(* IEC 61131-3 sources: Lasal/CPU_5344_V01/Class/RestartClass, 1 file *)

(* ---- RestartClass.st ---- *)
(*!
<Class
	Name               = "RestartClass"
	Revision           = "0.0"
	RealtimeTask       = "false"
	CyclicTask         = "false"
	BackgroundTask     = "false"
	Sigmatek           = "false"
	OSInterface        = "false"
	HighPriority       = "false"
	Automatic          = "false"
	UpdateMode         = "Prescan"
	SharedCommandTable = "true"
	Objectsize         = "(284,120)">
	<Channels>
		<Server Name="ClassSvr" Visualized="true" Initialize="false" WriteProtected="false" Retentive="false"/>
		<Client Name="os" Required="false" Internal="false"/>
	</Channels>
</Class>
*)
RestartClass : CLASS
  //Servers:
	ClassSvr 	: SvrChCmd_DINT;
  //Clients:
	os 	: CltChCmd__OSKernel;
  //Variables:
  //Functions:

	FUNCTION VIRTUAL GLOBAL ClassSvr::Write
		VAR_INPUT
			input (EAX) 	: DINT;
		END_VAR
		VAR_OUTPUT
			result (EAX) 	: DINT;
		END_VAR;
  //Tables:
	FUNCTION @STD
		VAR_OUTPUT
			ret_code	: CONFSTATES;
		END_VAR;
	FUNCTION GLOBAL TAB @CT_;
END_CLASS;

#pragma usingLtd _OSKernel

FUNCTION VIRTUAL GLOBAL RestartClass::ClassSvr::Write
	VAR_INPUT
		input (EAX) 	: DINT;
	END_VAR
	VAR_OUTPUT
		result (EAX) 	: DINT;
	END_VAR

	ClassSvr := input;

  os.Reboot();

	result := ClassSvr;

END_FUNCTION
